{attribute 'qualified_only'}
VAR_GLOBAL
	AMS_NETID				:STRING:='10.0.0.5.1.1';
	PROJECT_DIR				:STRING:='C:\250605-Aeromatic1\';
	DB_ID					:UDINT:=1;
	
	
	//Process constants
	GREASE_DENSITY			:REAL:=1;//[g/l]
	
	
	//Message IDs
	MSG_FillIntakeBuffer	:UINT := 10;
	
END_VAR

(* stored: Version 1.1.0.1
   GVL CONST: Id {7a4f5619-8a30-4379-b416-a1a7218e0288} *)
